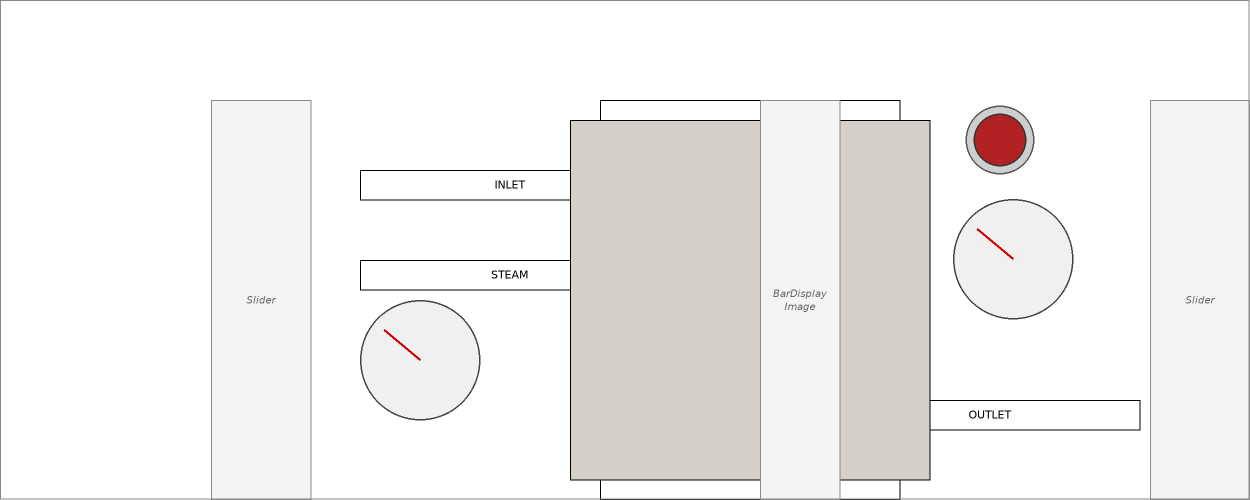
VISUALIZATION Vis  // 1250x500
    Rectangle (840,400 300x30), "OUTLET"
    Rectangle (360,170 300x30), "INLET"
    Rectangle (360,260 300x30), "STEAM"
    Rectangle (600,100 300x400)
    RoundedRectangle (570,120 360x360)
    BarDisplayImage (760,100 80x400), value: GVL.volPC_now, style: BarDisplayImage-Gray, scale format: %2d, scale 0..100
        p518627256: %
    Lamp1 (960,100 80x80), style: Lamp-Lamp1-Red
    Slider (1150,100 100x400), variable: GVL.valve_oule, scale 0..1
    Slider (211,100 100x400), variable: GVL.steam_temp, scale 0..100
    Meter360 (360,300 120x120), value: GVL.steam_temp, style: Meter-Meter360-Gray, scale format: %.1f, scale 0..100
    Meter360 (953,199 120x120), value: GVL.temp_now, style: Meter-Meter360-Gray, scale format: %.1f, scale 0..120
END_VISUALIZATION

(* stored: Version 1.1.0.1, ProductVersion 3.1.4024.12
   Visu Vis: Id {01a1e5c5-a279-4e0c-8b1a-faa13baf463d} *)
